# EPICS autosave request: 3-0/iocBoot/iocAMC100Test/AMC100Test_positions.req
$(P)MTR1.DVAL
$(P)MTR2.DVAL
$(P)MTR3.DVAL
